INTERFACE ValueRead EXTENDS __SYSTEM.IQueryInterface

METHOD Get
VAR_INPUT
END_VAR
END_METHOD

END_INTERFACE

(* stored: Version 1.1.0.1, ProductVersion 3.1.4024.15
   Itf ValueRead: Id {a1041c65-021b-4dce-8116-28824fba3b5b}
   Method Get: Id {bcbdc575-c1a9-4b54-b3d9-1957ab36cce4} *)
